FUNCTION_BLOCK EL3311
VAR
	_io : EL3xx1_Data;
	{attribute addProperty Name "WcState"}
	_wcState : WcStateInputToggle;
	{attribute addProperty Name "Info data"}
	_infoData : InfoDataAds;
END_VAR

PROPERTY IO : REFERENCE TO EL3xx1_Data
GET
IO REF= _io;
END_GET
END_PROPERTY

PROPERTY WcState : REFERENCE TO WcStateInputToggle
GET
WcState REF= _wcState;
END_GET
END_PROPERTY

END_FUNCTION_BLOCK

(* stored: Version 1.1.0.1, ProductVersion 3.1.4024.9
   POU EL3311: Id {33cb5fe5-1880-0d3b-1663-6f5895bf17b8}, SpecialFunc None
   Property IO: Id {40df3c3a-1576-0a4c-23e5-48b12be652eb}
   Get Get: Id {97e32b48-082e-00dd-2592-95d31783457e}
   Property WcState: Id {bfa83c3d-c6e7-07be-2448-9f176263cbe0}
   Get Get: Id {ca8d931b-8ed4-078f-2aea-b80b476ae6f8} *)
